TYPE ST_EL3443_DPM_MUX_REAL :
STRUCT
    nSelector : UINT := E_EL3443_DPM_Phase.Error_INDEX_Not_Valid;
    fValueRef : REFERENCE TO REAL;
END_STRUCT
END_TYPE

(* stored: Version 1.1.0.1, ProductVersion 3.1.4024.4
   DUT ST_EL3443_DPM_MUX_REAL: Id {8879b2fd-404e-41ad-9a67-0326ae9e1edc} *)
